ABB RobotStudio station: Attempt.rsstn

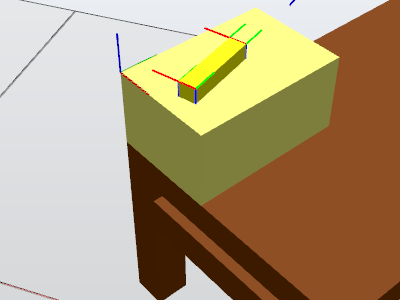
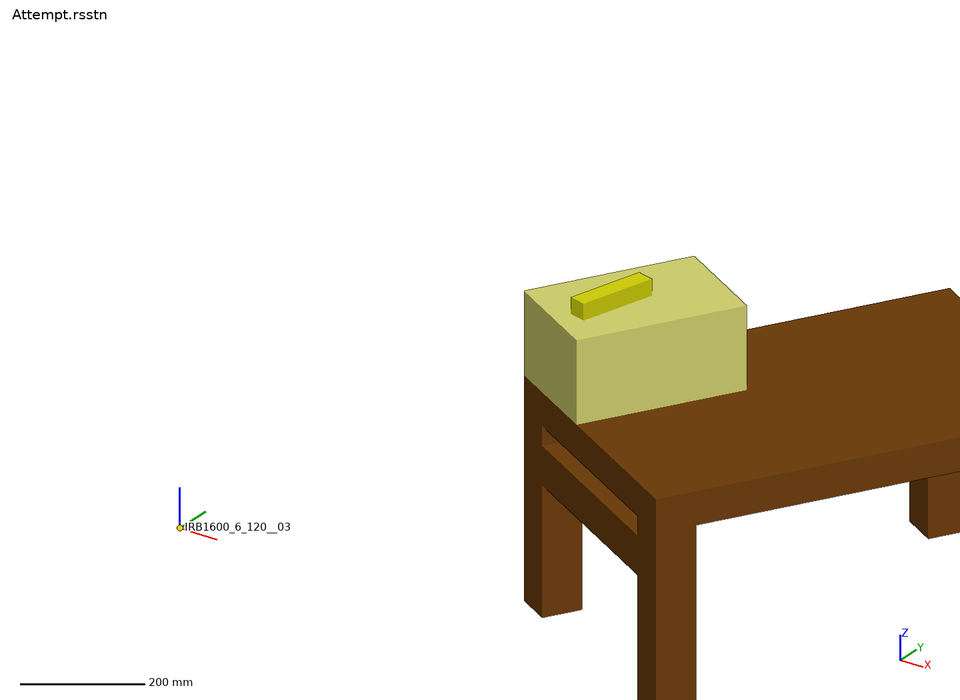
[picture v1: parts stored in the station drawn from their meshes, with robot base, taught points and paths (robot models come from the ABB library and are not in the file)]
Station Station (saved by RobotStudio 25.2.11266.1)
Controller Controller1
  mechanical unit ROB_1: IRB1600_6_120__03, 6 joints, base frame (0, 0, 0) mm
Layout (positions relative to the parent item):
  - IRB1600_6_120__03 [mechanism, from %ABB.RobotStudio.Models.IRB1600%\IRB1600_6_120_G_03.rslib] at (0, 0, 0) mm; joint values [0.0335, 0.1069, -0.2413, -3.189, -0.6587, 3.1958] (rad or m)
  - Pen [mechanism, from Library\Pen.rslib] at (851.13, 26.63, 1006.66) mm, rotated rx -180 ry 60 rz -180 deg
  - IRC5_Control-Module [part, from %ABB.RobotStudio.Models.IRC5%\IRC5_Control-Module.rslib] at (-759.17, -894.97, 100) mm, rotated rx 90 ry 0 rz 90 deg
  - Table [part] at (600, 100, 0) mm, rotated rx 0 ry 0 rz -30 deg, size 500 x 750 x 400 mm
  - Box [part] at (600, 100, 400) mm, rotated rx 0 ry 0 rz -30 deg, size 200 x 300 x 180 mm
Attachment: Pen is attached to IRB1600_6_120__03 / Link6
Targets, tools, work objects and paths stored in the station, written as RAPID:
! task T_ROB1
MODULE CalibData
  PERS tooldata Pen_TCP:=[TRUE,[[110,0,140],[0.707106781,0,0.707106781,0]],[1,[10.7435139,0,140],[1,0,0,0],0,0,0]];
  TASK PERS wobjdata Wobj_Box:=[FALSE,TRUE,"",[[599.999783494,100.000125,550],[0.9659258,0,0,-0.258819143]],[[0,0,0],[1,0,0,0]]];
ENDMODULE

! task T_ROB1
MODULE Module1
  CONST robtarget Target_10:=[[103.446463924,177.777860178,30],[0,-0.130526293,0.991444848,0],[0,0,0,0],[9E+09,9E+09,9E+09,9E+09,9E+09,9E+09]];
  CONST robtarget Target_20:=[[72.510503038,169.594512816,30],[0,-0.130526293,0.991444848,0],[0,0,0,0],[9E+09,9E+09,9E+09,9E+09,9E+09,9E+09]];
  CONST robtarget Target_30:=[[108.824546102,32.316800767,30],[0,-0.130526293,0.991444848,0],[0,0,0,0],[9E+09,9E+09,9E+09,9E+09,9E+09,9E+09]];
  CONST robtarget Target_40:=[[139.760506988,40.50014813,30],[0,-0.130526293,0.991444848,0],[0,0,0,0],[9E+09,9E+09,9E+09,9E+09,9E+09,9E+09]];
ENDMODULE

